// TwinCAT 3 PLC project PID_AS7
// ProgramVersion: 3.1.4023.0
// libraries:
//   Tc2_Standard, * (Beckhoff Automation GmbH)
//   Tc2_System, * (Beckhoff Automation GmbH)
//   Tc3_Module, * (Beckhoff Automation GmbH)
// project tree:
//   DUTs/ PID_Parameter_Strukt.TcDUT, PT1T2_Parameter_Strukt.TcDUT, System_Modus_Enum.TcDUT
//   GVLs/ GVL_Real_Block.TcGVL
//   / PlcTask.TcTTO
//   POUs/ F_VOLTAGE_TO_INT.TcPOU, MAIN.TcPOU, EncoderOverflow_RPMConversion.TcPOU, PID_Regler.TcPOU, PT1T2_Prozess.TcPOU
// real-time tasks:
//   TASK PlcTask: cycle T#1ms, priority 20, ADS port 350
// I/O:
//   DEVICE Device 1 (EtherCAT), AmsNetId 10.180.42.25.2.1
//     Term 1 (EK1200) [EK1200-5000 EtherCAT Power supply (2A E-Bus)]
//       Term 2 (EL1004) [EL1004 4Ch. Dig. Input 24V, 3ms]
//       Term 3 (EL2004) [EL2004 4Ch. Dig. Output 24V, 0.5A]
//       Term 4 (EL3004) [EL3004 4Ch. Ana. Input +/-10V]
//       Term 5 (EL4034) [EL4034 4Ch. Ana. Output +/-10V, 12bit]
//       Term 6 (EK1110) [EK1110 EtherCAT extension]
//     Term 7 (EK1100) [EK1100 EtherCAT Coupler (2A E-Bus)]
//       Term 8 (EL3004) [EL3004 4Ch. Ana. Input +/-10V]
//       Term 9 (EL5101) [EL5101 1Ch. Inc. Encoder 5V]
//       Term 10 (EL7342) [EL7342 2Ch. DC motor output stage (50V, 3.5A)]
//       Term 11 (EL9011) [EL9011 End Terminal]
// variable links:
//   PID_AS7/PID_AS7 Instance <-> Device 1 (EtherCAT)/Term 7 (EK1100)/Term 10 (EL7342)
//     PlcTask Outputs/GVL_Real_Block.motor_enable <-> DCM Control Channel 1/Control/Enable
//     PlcTask Outputs/GVL_Real_Block.motor_voltage <-> DCM Velocity Channel 1/Velocity
//   PID_AS7/PID_AS7 Instance <-> Device 1 (EtherCAT)/Term 7 (EK1100)/Term 9 (EL5101)
//     PlcTask Inputs/GVL_Real_Block.counter_overflow <-> ENC Status compact/Status/Counter overflow
//     PlcTask Inputs/GVL_Real_Block.counter_underflow <-> ENC Status compact/Status/Counter underflow
//     PlcTask Inputs/GVL_Real_Block.counter_value <-> ENC Status compact/Counter value

CONFIGURATION PID_AS7
    RESOURCE PLC ON TwinCAT3
        TASK PlcTask(INTERVAL := T#1ms, PRIORITY := 20);
        PROGRAM MAIN WITH PlcTask : MAIN;
    END_RESOURCE
END_CONFIGURATION

// ---- DUTs/PID_Parameter_Strukt.TcDUT
TYPE PID_Parameter_Strukt :
STRUCT
	K_p : REAL;		// Reglerverstärkung
	T_i : REAL;		// I-Anteil
	T_d : REAL; 	// D-Anteil
	N : UINT;		// D-Anteil Filterung
	ARW : BOOL;		// Anti-Reset Windup Aktiv
	u_min : REAL;	// Steuergrösse minimaler Wert
	u_max : REAL;	// Steuergrösse maximaler Wert
	Tr : REAL;		// ARW Faktor
END_STRUCT
END_TYPE

// ---- DUTs/PT1T2_Parameter_Strukt.TcDUT
TYPE PT1T2_Parameter_Strukt :
STRUCT
	K : REAL;
	T_1: REAL;
	T_2: REAL;
END_STRUCT
END_TYPE

// ---- DUTs/System_Modus_Enum.TcDUT
{attribute 'qualified_only'}
{attribute 'strict'}
TYPE System_Modus_Enum :
(
	enum_member := 0,
	System_Init,
	System_Run
);
END_TYPE

// ---- GVLs/GVL_Real_Block.TcGVL
{attribute 'qualified_only'}
VAR_GLOBAL
	counter_overflow AT %I* : BOOL;
	counter_underflow AT %I* : BOOL;
	counter_value AT %I* : UINT;
	motor_enable AT %Q* : BOOL;
	motor_voltage AT %Q* : INT;
	
END_VAR

// ---- POUs/MAIN.TcPOU
PROGRAM MAIN
VAR
	
	PT1T2Parameter : PT1T2_Parameter_Strukt;	// Parameter des Prozesses
	PID_Parameter : PID_Parameter_Strukt;
	Modus : System_Modus_Enum := System_Modus_Enum.System_Init;
	T : REAL;
	PID_1 : PID_Regler;
	PT1T2_1 : PT1T2_Prozess;
	ref : REAL;
	conversion_rpm : EncoderOverflow_RPMConversion;
	actual_rpm: REAL;
	initial_voltage: REAL := 0;
END_VAR

T := 0.001;		// Abtastzeit 1ms
GVL_Real_Block.motor_enable := TRUE;

GVL_Real_Block.motor_voltage := F_VOLTAGE_TO_INT(voltage := initial_voltage);
conversion_rpm(rpm_value => actual_rpm);




// Prozessparameter (PT1T2) definieren: Vollständig definiert
PT1T2_1.Param.K := 10;
PT1T2_1.Param.T_1 := 0.1;		// Ti = 10 * T
PT1T2_1.Param.T_2 := 0.01;		// Td = 0.1 * Ti

// Reglerparameter (PID)
PID_1.Param.K_p := 2.682;		//Kp 1/K, 10/K, 100/K
PID_1.Param.T_i := 1/55.34;
PID_1.Param.T_d := 0;
PID_1.Param.u_max := 24;					// Von Stellgrössen Limitierung gegeben
PID_1.Param.u_min := -24;						// Von Stellgrössen Limitierung gegeben
PID_1.Param.ARW := TRUE;					// Ein-/Ausschaltung Anti-Reset Windup

// Regler für DC-Motor implementieren
//PID_1(ref := ref, y := actual_rpm, Modus := Modus, Param := PID_1.Param, T := T, u_r => initial_voltage);

// A8 : Regelkreis implementieren
//PID_1(ref:= ref, y:= PT1T2_1.y_k, Modus := Modus, T := T);
//PT1T2_1(u := PID_1.u_r, Modus := Modus, T := T);

Modus := System_Modus_Enum.System_Run;


// 32767 fur +24 VDC und - 32767 fur -24VDC

END_PROGRAM

// ---- POUs/PID_Regler.TcPOU
FUNCTION_BLOCK PID_Regler
VAR_INPUT
	ref : REAL;						// Aktuelle Referenzgrösse (Soll-Grösse)
 	y : REAL;						// Aktuelle Regelgrösse (Ist-Grösse)
	Modus : System_Modus_Enum;		// Aktueller Modus (Init oder Run)
	Param : PID_Parameter_Strukt;	// Parameter der PID Reglers
	T : REAL;						// Abtastzeit
END_VAR
VAR_OUTPUT
	u_r : REAL;						// Stellgrösse Output
END_VAR
VAR
	u_k: REAL;						// P-Anteil des Reglers
	u_i_k: REAL;					// I-Anteil des Reglers
	u_d_k: REAL;					// D-Anteil des Reglers
	
	u_i_k_1: REAL;					// I-Anteil u_i[k-1]
	
	e_k: REAL;						// Fehler e_k := ref - y;
	e_k_1: REAL;					// Fehler e[k-1]
	
	i: REAL;						// Param.K_p / Param.T_i i-Faktor
	ad: REAL;						// Vorfaktor D-Anteil
	bd: REAL;						// Vorfaktor D-Anteil
	u_d_k_1: REAL;					// D-Anteil u_d[k-1]
	u_r_oS: REAL;					// u_r ohne Sättigung
	y_1: REAL;
END_VAR

// Repräsentiert den Regler

// CPU Belastung minimieren und soviel wie möglich schon im Init Modus berechnen
CASE Modus OF
	/// UNDEFINED ////
	System_Modus_Enum.enum_member:
		Modus := System_Modus_Enum.System_Init;
	
	/// INIT ///
	System_Modus_Enum.System_Init:
		i := Param.K_p / Param.T_i;
		Param.N := 10;
		ad := Param.T_d / (Param.T_d + Param.N * T);
		bd := (Param.K_p * Param.N * Param.T_d) / (Param.T_d + Param.N * T);
		Param.Tr := 0.001;
	
	/// RUN ///
	System_Modus_Enum.System_Run:
		e_k := ref - y;
		// A4: Diskretisiere den P-Anteil des analogen PID Reglers
		// Gibt keine andere Möglichkeit für u_k
		
		// P-Anteil
		u_k := Param.K_p * e_k;
		
		// A6: D-Anteil mit der Rückwärtsrechteckregel
		u_d_k := - (ad * u_d_k_1 + bd * (y - y_1));
		
		// Ohne Sättigung
		u_r_oS := u_k + u_i_k + u_d_k;
		
		// AS_8_A_1 Mit Saturation
		IF u_r_oS > param.u_max THEN
			u_r := Param.u_max;
		ELSIF u_r_oS < param.u_min THEN
			u_r := Param.u_min;
		ELSE
			// Sättigungsbereich nicht Erreicht und somit einfache Zuweisung
			u_r := u_r_oS;
		END_IF
		
		// Anti Reset (ARW) AS_8
		IF Param.ARW THEN
			// Mit Anti-Reset Windup. I-Anteil limitieren
			u_i_k := u_i_k_1 + i * ((e_k + e_k_1) / 2) * T + (T / Param.Tr) * (u_r - u_r_oS);
		ELSE
			// A5: Diskretisiere den I-Anteil des analogen PID Reglers mit Trapezregel (in Rek. Form)
			u_i_k := u_i_k_1 + i * ((e_k + e_k_1) / 2) * T;
		END_IF
		
		
		// Zuweisung alter Werte
		e_k_1 := e_k;
		u_d_k_1 := u_d_k;
		u_i_k_1 := u_i_k;
		y_1 := y;
		
	
END_CASE

END_FUNCTION_BLOCK

// ---- POUs/PT1T2_Prozess.TcPOU
FUNCTION_BLOCK PT1T2_Prozess
VAR_INPUT
	u : REAL;						// Aktuelle Steuergrösse
	Modus : System_Modus_Enum;		// Aktueller Modus(Init oder Run)
	Param : PT1T2_Parameter_Strukt;	// Parameter vom PT1T2 Modell
	T : REAL;						// Abtastzeit
END_VAR
VAR_OUTPUT
	y_k : REAL;
END_VAR
VAR
	b_0: REAL;
	b_1: REAL;
	c_1: REAL;
	c_2: REAL;
	
	a_1: REAL;
	a_2: REAL;
	
	y_k_1: REAL;
	y_k_2: REAL;
	u_k_1: REAL;
	u_k_2: REAL;
END_VAR

// Repräsentiert die Strecke

CASE Modus OF
	// Init Modus berechnet die Koeffizienten für H(z)
	System_Modus_Enum.System_Init:
		a_1 := EXP(-T/Param.T_1);
		a_2 := EXP(-T/Param.T_2);
		b_0 := Param.K/(Param.T_1 - Param.T_2)*(Param.T_1 * (1 - a_1)- Param.T_2 * ( 1 - a_2));
		b_1 := Param.K/(Param.T_1- Param.T_2)*(Param.T_2 * a_1 * (1 - a_2) - Param.T_1 * a_2 * (1 - a_1));
		c_1 := -(a_1 + a_2);
		c_2 := a_1 * a_2;

	// Run Modus implementiert die Differenzengleichung
	System_Modus_Enum.System_Run: 
		y_k := -c_1 * y_k_1 - c_2 * y_k_2 + b_0 * u_k_1 + b_1 * u_k_2;
		y_k_2 := y_k_1;
		y_k_1 := y_k;
		
		u_k_2 := u_k_1;
		u_k_1 := u;
		
		
END_CASE

END_FUNCTION_BLOCK

// ---- POUs/EncoderOverflow_RPMConversion.TcPOU
FUNCTION_BLOCK EncoderOverflow_RPMConversion

VAR_OUTPUT
	rpm_value: REAL; // RPM-Wert
END_VAR
VAR
	old_encoder_value: DINT := 0;
    rpm: REAL := 0.0;
    overflow: BOOL := FALSE;
	T : REAL := 0.001;
	edge_detected_overflow: BOOl;
	old_counter_overflow: BOOL := False;
	old_counter_underflow: BOOL;
	factor : REAL := 60 / (T*2048);
END_VAR

// detect rising edge of counter overflow. This means Encoder has reached maximum

// 1 rotation is 2048 Encoder Value
IF GVL_Real_Block.counter_overflow AND old_counter_overflow = FALSE THEN
	// Encoder Overflow detected counter_value starts again from zero
	rpm := DINT_TO_REAL((65535 - old_encoder_value) + GVL_Real_Block.counter_value) * factor;

    // rpm := LREAL_TO_REAL(0.0); // Setze RPM auf 0 bei einem Overflow
    // last_encoder_value := GVL_Real_Block.counter_value; // Aktualisiere den letzten Encoderwert
    // GVL_Real_Block.counter_overflow := FALSE; // Reset Overflow-Signal
ELSIF GVL_Real_Block.counter_underflow AND old_counter_underflow = FALSE THEN
	// Encoder Underflow detected counter_value new value ~65000
	rpm := DINT_TO_REAL(old_encoder_value + (65535 - GVL_Real_Block.counter_value)) * factor;

    //rpm := (UINT_TO_REAL(GVL_Real_Block.counter_value) - last_encoder_value)/T / 2048 * 60; // Umrechnung in RPM
    //last_encoder_value := GVL_Real_Block.counter_value; // Aktualisiere den letzten Encoderwert
ELSE
	// Normal without over/underflow
	rpm := DINT_TO_REAL(UINT_TO_DINT(GVL_Real_Block.counter_value) - old_encoder_value) * factor;
END_IF

old_counter_underflow := GVL_REAL_BLOCK.counter_underflow;
old_counter_overflow := GVL_Real_Block.counter_overflow;
old_encoder_value := GVL_Real_Block.counter_value;
rpm_value := rpm; // Aktualisiere den RPM-Wert

END_FUNCTION_BLOCK

// ---- POUs/F_VOLTAGE_TO_INT.TcPOU
FUNCTION F_VOLTAGE_TO_INT : INT
VAR_INPUT
	voltage : REAL;
END_VAR
VAR
	max_voltage : REAL := 24; // Maximum is 24V
	converted_value: INT;
END_VAR

IF voltage > max_voltage THEN
	voltage := max_voltage;
END_IF

IF voltage <= -max_voltage THEN
	voltage := -max_voltage;
END_IF

// Conversion expected GVL_Real_Block.motor_voltage within [1000 until -1000 from 0 on]
converted_value := REAL_TO_INT(32767 / max_voltage * voltage);

IF converted_value >= 32767 THEN
	F_VOLTAGE_TO_INT := 32767;

ELSIF converted_value <= -32767 THEN
	F_VOLTAGE_TO_INT := -32767;
ELSE
	F_VOLTAGE_TO_INT := converted_value;
END_IF

// 32767 fur +24 VDC und - ¨32767 fur -24VDC

END_FUNCTION
